TYPE T_Ctrl_SIf_ICL_In:
STRUCT
END_STRUCT
END_TYPE

(* stored: Version 1.1.0.1, ProductVersion 3.1.0.19
   DUT T_Ctrl_SIf_ICL_In: Id {2d45ca0a-5a20-4df3-84f1-a4654be1a830} *)
